{attribute 'qualified_only'}
{attribute 'strict'}
TYPE EOperationResult :
(
	none := 0,
	success := 1,
	busy := 2,
	recovering := 3,
	waiting := 4,
	failed := 5
);
END_TYPE

(* stored: Version 1.1.0.1, ProductVersion 3.1.4024.12
   DUT EOperationResult: Id {404ad134-b0d5-4c87-89ed-e088f9448317} *)
